// Mitsubishi GX Works2 project: solvvNpress_1   PLC: Q03UDV

PROGRAM MAIN
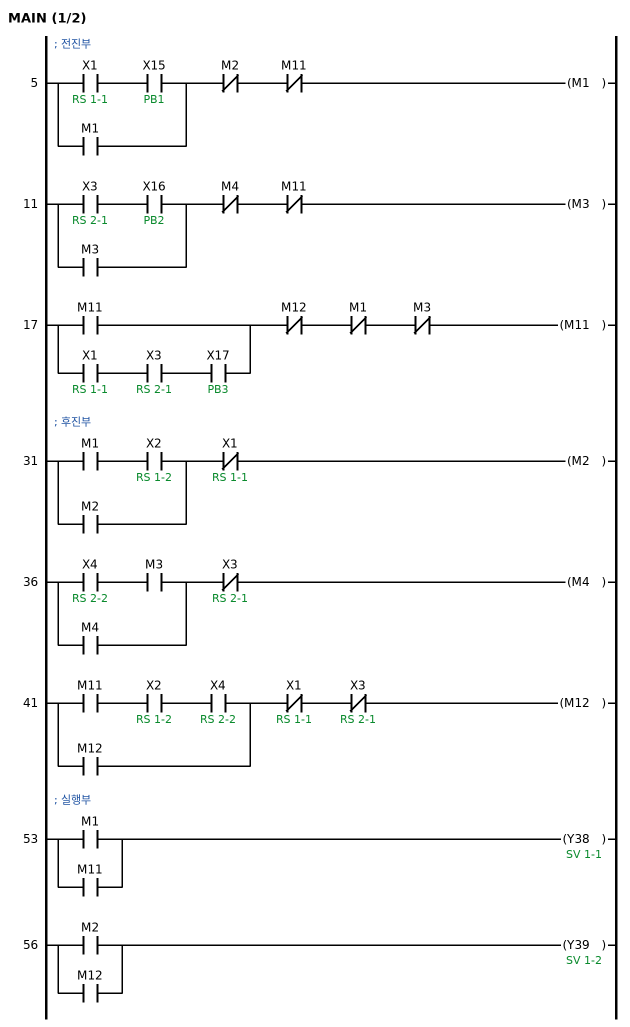
; 전진부
5     LD      X1  ; RS 1-1
      AND     X15  ; PB1
      OR      M1
      ANI     M2
      ANI     M11
      OUT     M1
11    LD      X3  ; RS 2-1
      AND     X16  ; PB2
      OR      M3
      ANI     M4
      ANI     M11
      OUT     M3
17    LD      M11
      LD      X1  ; RS 1-1
      AND     X3  ; RS 2-1
      AND     X17  ; PB3
      ORB
      ANI     M12
      ANI     M1
      ANI     M3
      OUT     M11
; 후진부
31    LD      M1
      AND     X2  ; RS 1-2
      OR      M2
      ANI     X1  ; RS 1-1
      OUT     M2
36    LD      X4  ; RS 2-2
      AND     M3
      OR      M4
      ANI     X3  ; RS 2-1
      OUT     M4
41    LD      M11
      AND     X2  ; RS 1-2
      AND     X4  ; RS 2-2
      OR      M12
      ANI     X1  ; RS 1-1
      ANI     X3  ; RS 2-1
      OUT     M12
; 실행부
53    LD      M1
      OR      M11
      OUT     Y38  ; SV 1-1
56    LD      M2
      OR      M12
      OUT     Y39  ; SV 1-2
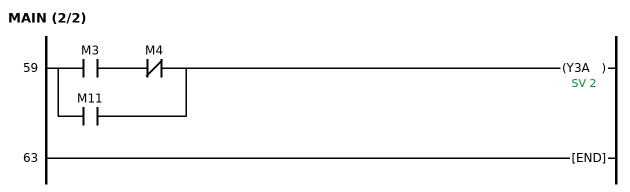
59    LD      M3
      ANI     M4
      OR      M11
      OUT     Y3A  ; SV 2
63    END
END_PROGRAM

// device comments not shown above
X18  ; PB4
Y30  ; LAMP1
Y31  ; LAMP2
Y3B  ; SV 3
